{attribute addProperty BoxType "ELM2642-0000-0016"}
{attribute addProperty Id "DO_Inputs_DeviceAT %I*DO_Inputs_Device_7B636AA11620DO_Group_1_OutputsAT %Q*DO_Group_1_Outputs_B15D14A01620DO_Group_2_OutputsAT %Q*DO_Group_2_Outputs_1AE88CA61620WcStateAT %I*WcState_98A4DF7520.250InfoDataAT %I*InfoData_0BDED7BF144180"}
{attribute addProperty CRC "3853189695"}
{attribute addProperty SizeInBites "194"}
{attribute addProperty SizeInBytes "24.25"}
TYPE ELM2642_A0E93795 :
STRUCT
	{attribute addProperty Name "DO_Inputs_Device"}
	DO_Inputs_Device : DO_Inputs_Device_7B636AA1;
	{attribute addProperty Name "DO_Group_1_Outputs"}
	DO_Group_1_Outputs : DO_Group_1_Outputs_B15D14A0;
	{attribute addProperty Name "DO_Group_2_Outputs"}
	DO_Group_2_Outputs : DO_Group_2_Outputs_1AE88CA6;
	{attribute addProperty Name "WcState"}
	WcState : WcState_98A4DF75;
	{attribute addProperty Name "InfoData"}
	InfoData : InfoData_0BDED7BF;
END_STRUCT
END_TYPE

(* stored: Version 1.2.0.0, ProductVersion 3.1.4024.9
   DUT ELM2642_A0E93795: Id {0f7a8e28-8cc3-4356-883d-42b33a3f72ba} *)
